(* PLC project KinIn_v3.project, CODESYS CODESYS V3.5 SP19 *)
(* stored: creationDateTime 2025-01-20T16:25:45.809065, modificationDateTime 2025-01-20T16:17:39.6822999 *)

FUNCTION_BLOCK se3ToSpatialVel
  VAR_INPUT
    se3mat : ARRAY[1..4, 1..4] OF REAL;
  END_VAR
  VAR_OUTPUT
    V : ARRAY[1..6] OF REAL;
  END_VAR

            V[1]:=se3mat[3, 2];
V[2]:=se3mat[1, 3];
V[3]:=se3mat[2, 1];
V[4]:=se3mat[1, 4];
V[5]:=se3mat[2, 4];
V[6]:=se3mat[3, 4];

          
END_FUNCTION_BLOCK
